FUNCTION_BLOCK BLOCK_STEP_TIMER
VAR_INPUT
	I_ON:					BOOL;
	PRM_TIME:				DINT;
	OP_RUN:					BLOCK_G7;				(*Grafcet de gestion de l'étape timer*)
	I_ROTATION_OK:			BOOL;					(*Condition rotation ok*)
	I_STOP_ROT_PS_OK:		BOOL;					(*Retour rotation PS à l'arrêt*)
	I_NO_ROTATION_PS:		BOOL;					(*Pas de rotation PS si consigne nulle*)
END_VAR
VAR_OUTPUT
	RQ_ROTATION_PS:			BOOL;
	RQ_STOP_ROTATION_PS:	BOOL;
	STATE_OK:				BOOL;
END_VAR
VAR
	FM_ETAPE1:		R_TRIG;
	FM_ETAPE2:		R_TRIG;
	FM_ETAPE3:		R_TRIG;
	FM_ETAPE4:		R_TRIG;
	TIMER:					TON;
END_VAR

FM_ETAPE1(CLK:=OP_RUN.Etape.1);
FM_ETAPE2(CLK:=OP_RUN.Etape.2);
FM_ETAPE3(CLK:=OP_RUN.Etape.3);
FM_ETAPE4(CLK:=OP_RUN.Etape.4);


RQ_ROTATION_PS:= FM_ETAPE1.Q AND NOT I_NO_ROTATION_PS;
RQ_STOP_ROTATION_PS := (FM_ETAPE1.Q AND I_NO_ROTATION_PS) OR FM_ETAPE3.Q;

TIMER( PT:= DINT_TO_TIME(PRM_TIME*1000),
		IN:=OP_RUN.Etape.2);
		
STATE_OK := OP_RUN.OK;

RUN_STEP();

ACTION RUN_STEP:
(*GRAFCET ETAPE EFFLUVAGE*)
(* initialisation du grafcet*)
OP_RUN(
	N_STEP_OP_OK:=4 ,
	N_STEP_OP_NOK:= 0);

(* initialisation du grafcet*)
IF 		OP_RUN.Etape = 0 THEN
				OP_RUN.Etape.0 := TRUE;
(*repositionnement sur étape 0*)
ELSIF  NOT I_ON THEN
		OP_RUN.Etape:= 0;			(*RAZ grafcet*)
		OP_RUN.Etape.0:= TRUE;
(*étape 0-1 *)
ELSIF OP_RUN.Etape.0 AND I_ON  THEN
		OP_RUN.Etape.1 	:= TRUE;
		OP_RUN.Etape.0 	:= FALSE;
(*étape 2-1*)
ELSIF OP_RUN.Etape.1 AND ((I_ROTATION_OK AND NOT I_NO_ROTATION_PS) OR (I_STOP_ROT_PS_OK AND I_NO_ROTATION_PS)) THEN
		OP_RUN.Etape.2 	:= TRUE;
		OP_RUN.Etape.1 	:= FALSE;
(*étape 2-3*)
ELSIF OP_RUN.Etape.2 AND TIMER.Q THEN 
		OP_RUN.Etape.3	:= TRUE;
		OP_RUN.Etape.2	:= FALSE;
(*étape 3-4*)
ELSIF OP_RUN.Etape.3 AND I_STOP_ROT_PS_OK THEN 
		OP_RUN.Etape.4	:= TRUE;
		OP_RUN.Etape.3	:= FALSE;
END_IF

OP_RUN.POST();
END_ACTION

END_FUNCTION_BLOCK

(* stored: Version 1.1.0.1, ProductVersion 3.1.4024.11
   POU BLOCK_STEP_TIMER: Id {4e4b1079-1279-4786-a479-f5115f4016f9}, SpecialFunc None
   Action RUN_STEP: Id {f91ab6c2-d249-4020-a9b8-d24bc409f6ff} *)
